FUNCTION F_LogLA3C 
VAR_INPUT
	eLogLevel		: E_LogLevel;
	sLogger			: T_MaxString;
	sMessage		: T_MaxString;
	aArg1			: ANY;
	aArg2			: ANY;
	aArg3			: ANY;
	iContextBuilder	: I_ContextBuilder;
END_VAR
VAR 
	aEmptyArg		: BYTE;
END_VAR

F_LogA(
	eLogLevel,
	sLogger,
	sMessage,
	3,
	aArg1,
	aArg2,
	aArg3,
	aEmptyArg,
	aEmptyArg,
	aEmptyArg,
	aEmptyArg,
	aEmptyArg,
	aEmptyArg,
	aEmptyArg,
	iContextBuilder
);

END_FUNCTION

(* stored: Version 1.1.0.1, ProductVersion 3.1.4024.0
   POU F_LogLA3C: Id {517c391a-d776-4625-84c0-0556794529da}, SpecialFunc None *)
